% RSLogix 500 project demorgan_puzzle_202012.RSS, saved by version 8.30.00.16 %
PROJECT "UNTITLED"    % processor: Bul.1763 MicroLogix 1100 Series B %

PROGRAM FILES
  LAD 2   5 rungs

DATA FILES
  O0 OUTPUT  4 elements
  I1 INPUT  6 elements
  S2 STATUS  66 elements
  B3 BINARY  1 elements
  T4 TIMER  1 elements
  C5 COUNTER  3 elements
  R6 CONTROL  1 elements
  N7 INTEGER  4 elements
  F8 FLOAT  1 elements

LADDER 2
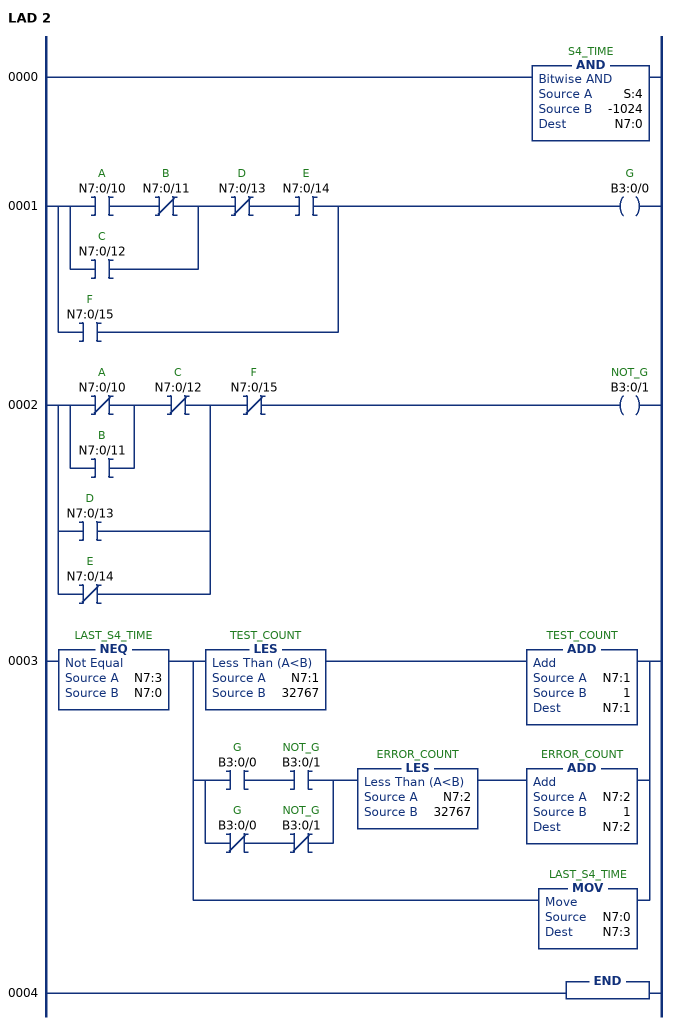
% Rung: 0 %
SOR AND S:4 -1024 N7:0 EOR
%   S:4  "Time Base" %
%   N7:0  S4_TIME %
% Rung: 1 %
SOR BST BST XIC N7:0/10 XIO N7:0/11 NXB XIC N7:0/12 BND XIO N7:0/13 XIC N7:0/14 NXB XIC N7:0/15 BND OTE B3:0/0 EOR
%   N7:0/10  A %
%   N7:0/11  B %
%   N7:0/12  C %
%   N7:0/13  D %
%   N7:0/14  E %
%   N7:0/15  F %
%   B3:0/0  G %
% Rung: 2 %
SOR BST BST XIO N7:0/10 NXB XIC N7:0/11 BND XIO N7:0/12 NXB XIC N7:0/13 NXB XIO N7:0/14 BND XIO N7:0/15 OTE B3:0/1 EOR
%   N7:0/10  A %
%   N7:0/11  B %
%   N7:0/12  C %
%   N7:0/13  D %
%   N7:0/14  E %
%   N7:0/15  F %
%   B3:0/1  NOT_G %
% Rung: 3 %
SOR NEQ N7:3 N7:0 BST LES N7:1 32767 ADD N7:1 1 N7:1 NXB BST XIC B3:0/0 XIC B3:0/1 NXB XIO B3:0/0 XIO B3:0/1 BND LES N7:2 32767 ADD N7:2 1 N7:2 NXB MOV N7:0 N7:3 BND EOR
%   N7:3  LAST_S4_TIME %
%   N7:0  S4_TIME %
%   N7:1  TEST_COUNT %
%   B3:0/0  G %
%   B3:0/1  NOT_G %
%   N7:2  ERROR_COUNT %
% Rung: 4 %
SOR END EOR

DATA TABLE (non-zero values as saved)
DATA T4
% .PRE .ACC %
% T4:0 % 200 0
DATA C5
% .PRE .ACC %
% C5:0 % 32767 24
% C5:1 % 32767 12
% C5:2 % 32767 12
DATA R6
% .LEN .POS %
% R6:0 % 8 4
DATA N7
% N7:0 % 0 0 0 -1
DATA F8
% F8:0 % 10188
